PROGRAM Ax_01_AxisSpeedSelect_03
VAR
	HMI_Motion: FB_HMI_Control_NoGroupRef;


	tMessageOffset: UINT;
	tNumMessagesPerRow: UINT;
	
	
	MyAdvanceInterlock: BOOL;
	MyReturnInterlock: BOOL;
	
	MyAutoAdvanceCondition: BOOL;
	MyAutoReturnCondition: BOOL;
	
	myAdvancePrompt: BOOL;
	myReturnPrompt: BOOL;
	

	NotUsed: UINT;
	
	selection :INT;
	
END_VAR
VAR // added by the converter: edge detectors and wires of the graphical bodies
    _w1 : BOOL;
    _rt1, _rt2 : R_TRIG;
END_VAR

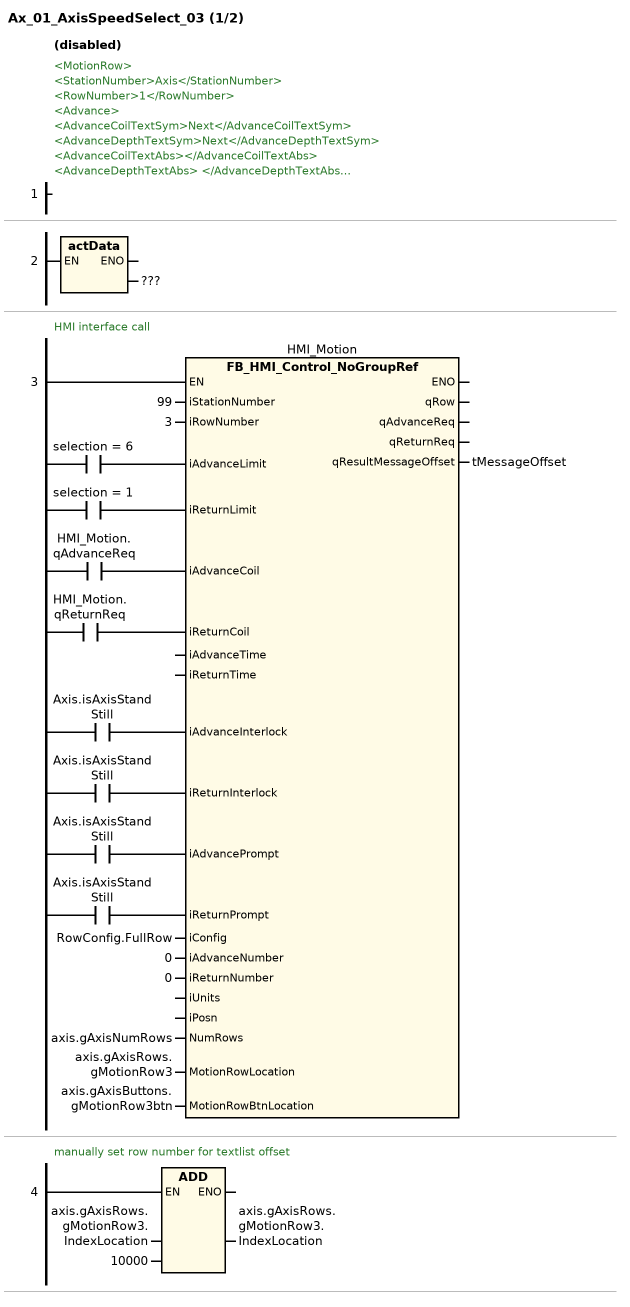
// NETWORK 1 (disabled)
// <MotionRow>
// <StationNumber>Axis</StationNumber>
// <RowNumber>1</RowNumber>
//   <Advance>
//     <AdvanceCoilTextSym>Next</AdvanceCoilTextSym>
//     <AdvanceDepthTextSym>Next</AdvanceDepthTextSym>
//     <AdvanceCoilTextAbs></AdvanceCoilTextAbs>
//     <AdvanceDepthTextAbs> </AdvanceDepthTextAbs>
//     <ManSeq></ManSeq>
//   </Advance>
//   <Return>
//     <ReturnCoilTextSym>Previous</ReturnCoilTextSym>
//     <ReturnDepthTextSym>Previous</ReturnDepthTextSym>
//     <ReturnCoilTextAbs></ReturnCoilTextAbs>
//     <ReturnDepthTextAbs></ReturnDepthTextAbs>
//    <ManSeq></ManSeq>
//   </Return>
//   <Motion>
//     <NameSym>Axis Name</NameSym>
//     <NameAbs>X1</NameAbs>
//   </Motion>
// </MotionRow>

// NETWORK 2
actData();

// NETWORK 3
// HMI interface call
HMI_Motion(
    iStationNumber := 99,
    iRowNumber := 3,
    iAdvanceLimit := selection = 6,
    iReturnLimit := selection = 1,
    iAdvanceCoil := HMI_Motion.qAdvanceReq,
    iReturnCoil := HMI_Motion.qReturnReq,
    iAdvanceInterlock := Axis.isAxisStandStill,
    iReturnInterlock := Axis.isAxisStandStill,
    iAdvancePrompt := Axis.isAxisStandStill,
    iReturnPrompt := Axis.isAxisStandStill,
    iConfig := RowConfig.FullRow,
    iAdvanceNumber := 0,
    iReturnNumber := 0,
    NumRows := axis.gAxisNumRows,
    MotionRowLocation := axis.gAxisRows.gMotionRow3,
    MotionRowBtnLocation := axis.gAxisButtons.gMotionRow3btn,
    qResultMessageOffset => tMessageOffset); // FB_HMI_Control_NoGroupRef

// NETWORK 4
// manually set row number for textlist offset
axis.gAxisRows.gMotionRow3.IndexLocation := axis.gAxisRows.gMotionRow3.IndexLocation + 10000;

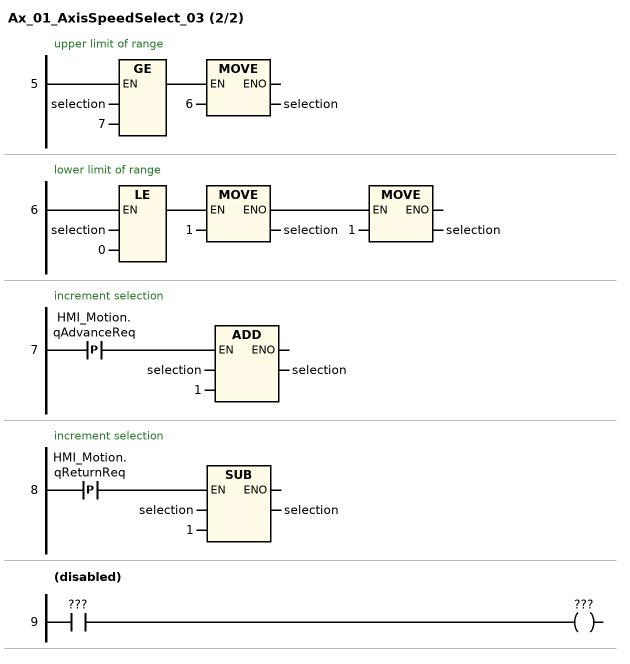
// NETWORK 5
// upper limit of range
IF selection >= 7 THEN selection := 6; END_IF

// NETWORK 6
// lower limit of range
_w1 := selection <= 0;
IF _w1 THEN selection := 1; END_IF
IF _w1 THEN selection := 1; END_IF

// NETWORK 7
// increment selection
_rt1(CLK := HMI_Motion.qAdvanceReq);
IF _rt1.Q THEN selection := selection + 1; END_IF

// NETWORK 8
// increment selection
_rt2(CLK := HMI_Motion.qReturnReq);
IF _rt2.Q THEN selection := selection - 1; END_IF

// NETWORK 9 (disabled)
// ??? := ???;

ACTION actData:
//move data from axis. data to the HMI for viewing on the motionRows


CASE selection OF
	1:
		HMI_Motion.iPosn := '0.1';
	2:
		HMI_Motion.iPosn := '1';
	3:
		HMI_Motion.iPosn := '5';
	4:
		HMI_Motion.iPosn := '10.0';
	5:
		HMI_Motion.iPosn := '25.0';
	6:
		HMI_Motion.iPosn := '100.0';
			
END_CASE



IF axis.axisSelected.isLinearDrive THEN
	HMI_Motion.iUnits := ' mm/s';
END_IF

IF axis.axisSelected.isSpindleDrive THEN
	HMI_Motion.iUnits := ' deg/s';
END_IF
END_ACTION

END_PROGRAM

(* stored: Version 1.1.0.1, ProductVersion 3.1.4024.12
   POU Ax_01_AxisSpeedSelect_03: Id {0469215d-e5f1-44a0-bcb4-c71d7d6b3479}, SpecialFunc None
   Action actData: Id {770c7a07-28f1-4fd2-b299-f3605f58c502} *)
